// TIA Portal V18 export
// export: Created 2026-06-08T16:32:21.3714393Z, ExportSetting WithDefaults, DisplayName Totally Integrated Automation Portal, DisplayVersion V18, DisplayName TIA Portal Openness, DisplayVersion V18, DisplayName TIA Portal Version Control Interface, DisplayVersion V18, DisplayName STEP 7 Professional, DisplayVersion V18, DisplayName STEP 7 Safety, DisplayVersion V18, DisplayName WinCC Professional, DisplayVersion V18
FUNCTION_BLOCK "Assembly_Green"   // FB10, LAD
VERSION : 0.1
// stored: AutoNumber true, IsIECCheckEnabled false, UDAEnableTagReadback false
   VAR_TEMP   // added for the SCL form of the ladder/FBD networks
      _w1 : Bool;
      _s5time1 : S5Time;
   END_VAR
BEGIN

REGION Network 1
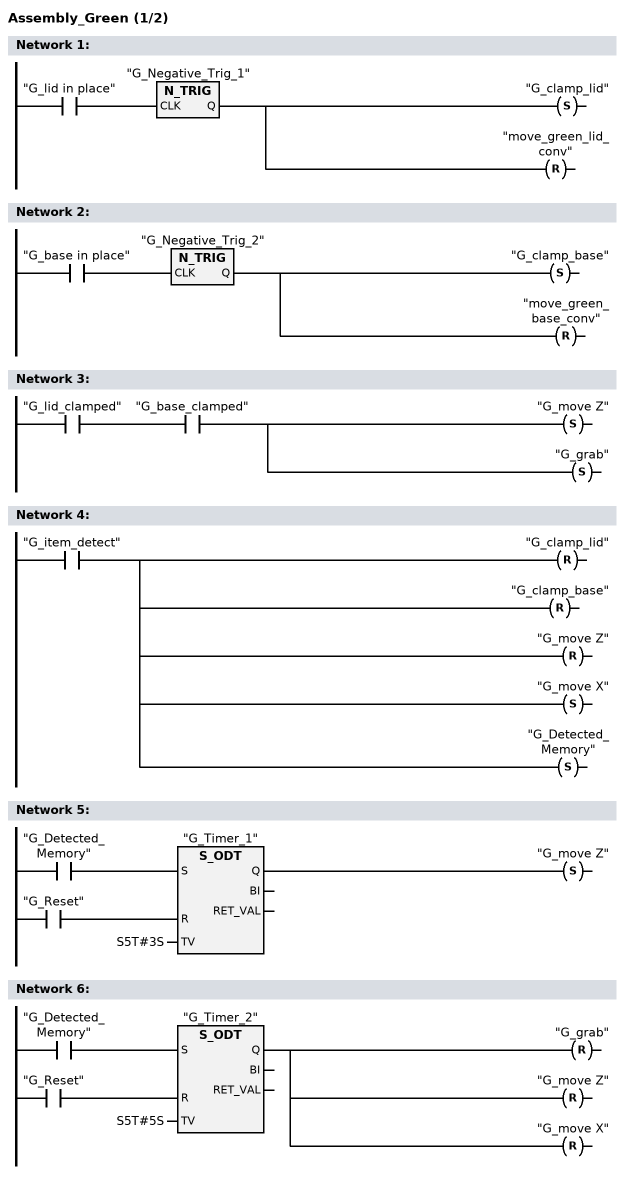
   RUNG wire#powerrail
      Contact( "G_lid in place" )
      N_Trig( "G_Negative_Trig_1" )
      wire#w1
      S_Coil( "G_clamp_lid" )
   END_RUNG
   RUNG wire#w1
      R_Coil( "move_green_lid_conv" )
   END_RUNG
   // the same network as SCL:
   #_w1 := NOT "G_lid in place" AND "G_Negative_Trig_1";   // falling edge
   "G_Negative_Trig_1" := "G_lid in place";
   IF #_w1 THEN
       "G_clamp_lid" := TRUE;
       "move_green_lid_conv" := FALSE;
   END_IF;
END_REGION

REGION Network 2
   RUNG wire#powerrail
      Contact( "G_base in place" )
      N_Trig( "G_Negative_Trig_2" )
      wire#w1
      S_Coil( "G_clamp_base" )
   END_RUNG
   RUNG wire#w1
      R_Coil( "move_green_base_conv" )
   END_RUNG
   // the same network as SCL:
   #_w1 := NOT "G_base in place" AND "G_Negative_Trig_2";   // falling edge
   "G_Negative_Trig_2" := "G_base in place";
   IF #_w1 THEN
       "G_clamp_base" := TRUE;
       "move_green_base_conv" := FALSE;
   END_IF;
END_REGION

REGION Network 3
   RUNG wire#powerrail
      Contact( "G_lid_clamped" )
      Contact( "G_base_clamped" )
      wire#w1
      S_Coil( "G_move Z" )
   END_RUNG
   RUNG wire#w1
      S_Coil( "G_grab" )
   END_RUNG
   // the same network as SCL:
   IF "G_lid_clamped" AND "G_base_clamped" THEN
       "G_move Z" := TRUE;
       "G_grab" := TRUE;
   END_IF;
END_REGION

REGION Network 4
   RUNG wire#powerrail
      Contact( "G_item_detect" )
      wire#w1
      R_Coil( "G_clamp_lid" )
   END_RUNG
   RUNG wire#w1
      R_Coil( "G_clamp_base" )
   END_RUNG
   RUNG wire#w1
      R_Coil( "G_move Z" )
   END_RUNG
   RUNG wire#w1
      S_Coil( "G_move X" )
   END_RUNG
   RUNG wire#w1
      S_Coil( "G_Detected_Memory" )
   END_RUNG
   // the same network as SCL:
   IF "G_item_detect" THEN
       "G_clamp_lid" := FALSE;
       "G_clamp_base" := FALSE;
       "G_move Z" := FALSE;
       "G_move X" := TRUE;
       "G_Detected_Memory" := TRUE;
   END_IF;
END_REGION

REGION Network 5
   RUNG wire#powerrail
      Contact( "G_Detected_Memory" )
      S_ODT(T_NO := "G_Timer_1", R := wire#w1, TV := S5T#3S, BI =>, RET_VAL =>)
      S_Coil( "G_move Z" )
   END_RUNG
   RUNG wire#powerrail
      Contact( "G_Reset" )
   END_RUNG wire#w1
   // the same network as SCL:
   #_s5time1 := S_ODT(T_NO := "G_Timer_1", S := "G_Detected_Memory", R := "G_Reset", TV := S5T#3S, Q => #_w1);
   IF #_w1 THEN "G_move Z" := TRUE; END_IF;
END_REGION

REGION Network 6
   RUNG wire#powerrail
      Contact( "G_Detected_Memory" )
      S_ODT(T_NO := "G_Timer_2", R := wire#w1, TV := S5T#5S, BI =>, RET_VAL =>)
      wire#w2
      R_Coil( "G_grab" )
   END_RUNG
   RUNG wire#powerrail
      Contact( "G_Reset" )
   END_RUNG wire#w1
   RUNG wire#w2
      R_Coil( "G_move Z" )
   END_RUNG
   RUNG wire#w2
      R_Coil( "G_move X" )
   END_RUNG
   // the same network as SCL:
   #_s5time1 := S_ODT(T_NO := "G_Timer_2", S := "G_Detected_Memory", R := "G_Reset", TV := S5T#5S, Q => #_w1);
   IF #_w1 THEN
       "G_grab" := FALSE;
       "G_move Z" := FALSE;
       "G_move X" := FALSE;
   END_IF;
END_REGION

REGION Network 7
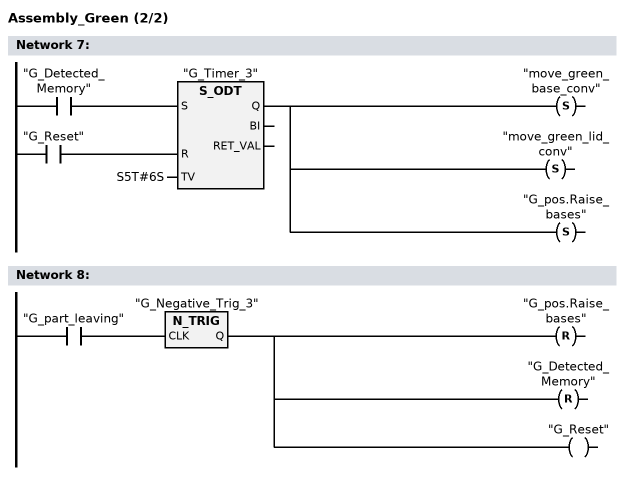
   RUNG wire#powerrail
      Contact( "G_Detected_Memory" )
      S_ODT(T_NO := "G_Timer_3", R := wire#w1, TV := S5T#6S, BI =>, RET_VAL =>)
      wire#w2
      S_Coil( "move_green_base_conv" )
   END_RUNG
   RUNG wire#powerrail
      Contact( "G_Reset" )
   END_RUNG wire#w1
   RUNG wire#w2
      S_Coil( "move_green_lid_conv" )
   END_RUNG
   RUNG wire#w2
      S_Coil( "G_pos.Raise_bases" )
   END_RUNG
   // the same network as SCL:
   #_s5time1 := S_ODT(T_NO := "G_Timer_3", S := "G_Detected_Memory", R := "G_Reset", TV := S5T#6S, Q => #_w1);
   IF #_w1 THEN
       "move_green_base_conv" := TRUE;
       "move_green_lid_conv" := TRUE;
       "G_pos.Raise_bases" := TRUE;
   END_IF;
END_REGION

REGION Network 8
   RUNG wire#powerrail
      Contact( "G_part_leaving" )
      N_Trig( "G_Negative_Trig_3" )
      wire#w1
      R_Coil( "G_pos.Raise_bases" )
   END_RUNG
   RUNG wire#w1
      R_Coil( "G_Detected_Memory" )
   END_RUNG
   RUNG wire#w1
      Coil( "G_Reset" )
   END_RUNG
   // the same network as SCL:
   #_w1 := NOT "G_part_leaving" AND "G_Negative_Trig_3";   // falling edge
   "G_Negative_Trig_3" := "G_part_leaving";
   IF #_w1 THEN
       "G_pos.Raise_bases" := FALSE;
       "G_Detected_Memory" := FALSE;
   END_IF;
   "G_Reset" := #_w1;
END_REGION
END_FUNCTION_BLOCK
